FUNCTION_BLOCK RobotA21_1 EXTENDS KukaRobot
VAR_OUTPUT //from outputs array
	{warning disable C0195}
	//taskID : A21;
	//param1 : INT;
	//param2 : INT;
	//Xmm : INT;
	//Ymm : INT;
	//Zmm : INT;
	//angle : INT;
	//stagingOccupancy : INT;
	//insertionSuctionStatus : INT;
	//magazineStatus : INT; //unused
	inspectionValue : INT;
	
	strapSafetyOut : BOOL;
END_VAR
VAR_OUTPUT //from inputs array
	tool : SectionEnum := SectionEnum.WOOD_BUNK;
	suspendedMaterial : STRING;
	//gripper : EOAT := (id := SectionEnum.WOOD_BUNK, material := '');
	
	completedTask : A21;
	eoatDistance : INT;
	woodBunkAvailability : INT;
	chipboardAvailability : INT;
	materialAtHoldingPosition : INT;
	
	strapSafetyIn : BOOL;
END_VAR
VAR
	reservationEnum : SectionEnum;
	hmiTask : STRING;
	hmiTool : STRING;
END_VAR
(*
extends KukaRobot
assigns descriptive labels to each IO group from the array
additional section-specific methods to get/set IO groups
*)

(*
parameters - aliases to IO elements
command - full IO array
*)
{warning disable C0195}
SUPER^();

strapSafetyOut := NOT strapperA21.enable AND NOT strapperA21.execute;
outputs[8].15 := strapSafetyOut;

outputs[1] := taskID;
outputs[2] := param1;
outputs[3] := param2;
outputs[4] := Xmm;
outputs[5] := Ymm;
outputs[6] := Zmm;
outputs[7] := angle;
outputs[8] := stagingOccupancy;
outputs[9] := insertionSuctionStatus;
outputs[10] := magazineStatus;
outputs[11] := inspectionValue;

outputs[8].15 := strapSafetyOut;

refreshParameters();

reservationEnum := reservation;
IF reservationEnum = SectionEnum.NULL_SECTION THEN
	hmiReservation := 'N/A';
ELSE
	hmiReservation := TO_STRING(reservationEnum);
END_IF

hmiTask := TO_STRING(taskID);
hmiTool := TO_STRING(tool);

{attribute 'monitoring' := 'call'}
PROPERTY Angle : INT
GET
END_GET
SET
END_SET
END_PROPERTY

{attribute 'monitoring' := 'call'}
PROPERTY Busy : BOOL
GET
VAR
	//emptyOutput : ARRAY[1..50] OF INT;
END_VAR
//Busy stays TRUE until outputs are cleared AND completed task has elapsed
//Ready is always inverse of Busy
refreshParameters();

Busy := taskID <> 0 OR completedTask <> 0;
END_GET
END_PROPERTY

METHOD changeEOAT : BOOL
VAR_INPUT
	targetTool : SectionEnum;
END_VAR
setGroup(group := 1, value := A21.TOOL_CHANGE_CHIPBOARD);
setGroup(group := 1, value := A21.TOOL_CHANGE_BUNK);

changeEOAT := tool = targetTool;
END_METHOD

METHOD clearCommand : BOOL
VAR_INPUT
END_VAR
SUPER^.clearCommand();

refreshParameters();
END_METHOD

{attribute 'monitoring' := 'call'}
PROPERTY Done : BOOL
GET
refreshParameters();

Done :=
	completedTask = taskID AND
	taskID <> 0 AND
	completedTask <> 0;
END_GET
END_PROPERTY

{attribute 'monitoring' := 'call'}
PROPERTY HoldMaterial : STRING
GET
HoldMaterial := suspendedMaterial;
END_GET
SET
suspendedMaterial := HoldMaterial;
END_SET
END_PROPERTY

{attribute 'monitoring' := 'call'}
PROPERTY Param1 : INT
GET
END_GET
SET
END_SET
END_PROPERTY

{attribute 'monitoring' := 'call'}
PROPERTY Param2 : INT
GET
END_GET
SET
END_SET
END_PROPERTY

{attribute 'monitoring' := 'call'}
PROPERTY Ready : BOOL
GET
refreshParameters();

Ready := taskID = 0 AND completedTask = 0;
END_GET
END_PROPERTY

METHOD PRIVATE refreshParameters : BOOL
VAR_INPUT
END_VAR
{warning disable C0196}
taskID := outputs[1];
param1 := outputs[2];
param2 := outputs[3];
Xmm := outputs[4];
Ymm := outputs[5];
Zmm := outputs[6];
angle := outputs[7];
stagingOccupancy := outputs[8];
insertionSuctionStatus := outputs[9];
magazineStatus := outputs[10]; //unused
inspectionValue := outputs[11];

completedTask := inputs[1];
eoatDistance := inputs[2];
woodBunkAvailability := inputs[3];
chipboardAvailability := inputs[4];
materialAtHoldingPosition := inputs[5];
//robotEOAT := inputs[6];

strapSafetyIn := inputs[4].15;
END_METHOD

METHOD setGroup : BOOL
VAR_INPUT
	group : INT;
	value : INT;
END_VAR
SUPER^.setGroup(group := group, value := value);

refreshParameters();
END_METHOD

METHOD setParameters : BOOL
VAR_INPUT
	newTaskID : INT;
	newParam1 : INT;
	newParam2 : INT;
	newXmm : INT;
	newYmm : INT;
	newZmm : INT;
	newAngle : INT;
	newStagingOccupancy : INT;
	newInsertionSuctionStatus : INT;
	newMagazineStatus : INT; //unused
	newInspectionValue : INT;
END_VAR
setGroup(group := 1, value := newTaskID);
setGroup(group := 2, value := newParam1);
setGroup(group := 3, value := newParam2);
setGroup(group := 4, value := newXmm);
setGroup(group := 5, value := newYmm);
setGroup(group := 6, value := newZmm);
setGroup(group := 7, value := newAngle);

newStagingOccupancy.15 := NOT strapperA21.enable AND NOT strapperA21.execute;
setGroup(group := 8, value := newStagingOccupancy);

setGroup(group := 9, value := newInsertionSuctionStatus);
setGroup(group := 10, value := newMagazineStatus);
setGroup(group := 11, value := newInspectionValue);

refreshParameters();
END_METHOD

{attribute 'monitoring' := 'call'}
PROPERTY StagingOccupancy : INT
GET
END_GET
SET
END_SET
END_PROPERTY

{attribute 'monitoring' := 'call'}
PROPERTY TaskID : A21
GET
TaskID := outputs[1];
END_GET
SET
outputs[1] := TaskID;
END_SET
END_PROPERTY

{attribute 'monitoring' := 'call'}
PROPERTY Xmm : INT
GET
END_GET
SET
END_SET
END_PROPERTY

{attribute 'monitoring' := 'call'}
PROPERTY Ymm : INT
GET
END_GET
SET
END_SET
END_PROPERTY

{attribute 'monitoring' := 'call'}
PROPERTY Zmm : INT
GET
END_GET
SET
END_SET
END_PROPERTY

END_FUNCTION_BLOCK

(* stored: Version 1.1.0.1, ProductVersion 3.1.4024.11
   POU RobotA21_1: Id {67986ee9-35d0-4991-b5f7-67f7ce42987a}, SpecialFunc None
   Folder Groups: Id {eb42e132-aba5-47c8-8cae-a23ba92d8609}
   Folder Outputs: Id {321cea36-5d8f-400f-a5af-fdd868e827da}
   Folder Parameters: Id {c3d578fe-defd-4b12-9c77-b5953ca5c70d}
   Folder Properties: Id {eb91b964-775c-4fcb-b72d-754eac110c77}
   Property Angle: Id {4e283426-00f0-4c6b-b031-919967f9904b}
   Get Get: Id {86ab762a-e94a-42de-be5d-1c1d6883e23c}
   Set Set: Id {d8c9edf3-2c7c-45ce-acf1-984193f826aa}
   Property Busy: Id {79b3ce6a-9c01-452d-bb4a-867892b7100d}
   Get Get: Id {d9f24df2-3a79-4dc5-8239-3effa750f19a}
   Method changeEOAT: Id {056c48cb-6b24-46e5-adc1-74bf302c5ce2}
   Method clearCommand: Id {9155dabb-946e-465d-83be-8bd2e505d8d8}
   Property Done: Id {9e7360cb-1f33-47df-8e4b-f7735364d7f4}
   Get Get: Id {93f104fb-aef5-4ea5-b5b3-4fe7369ec6e3}
   Property HoldMaterial: Id {496f148f-ed6a-4218-9fd8-2d6729172b93}
   Get Get: Id {f10adf07-73d8-475e-92ad-0736f496bafa}
   Set Set: Id {6785f88a-284f-4b38-9b72-c0d119fc1118}
   Property Param1: Id {65d5818f-490f-4753-a4a0-b72affe7ebe5}
   Get Get: Id {33c584a1-59b3-4725-9a29-2b55d6bca155}
   Set Set: Id {a24ce27a-d8c3-4182-8d2d-af3bc85cb9c6}
   Property Param2: Id {45986bf8-e408-4761-908a-a14fdd4e0c5f}
   Get Get: Id {00d89721-8515-4692-bbde-4208e35fdac9}
   Set Set: Id {c3ea74de-9992-4db6-afa9-9cbc7c3fbab9}
   Property Ready: Id {369f7773-2368-4d49-8b91-351e545a75a3}
   Get Get: Id {215529ad-6487-4575-a731-48e5f5ac5cf5}
   Method refreshParameters: Id {84265115-d663-44b8-b8b9-61681c9d0c6b}
   Method setGroup: Id {611ab68f-21d7-4b39-adf2-beaae57f94ff}
   Method setParameters: Id {1354b4cc-1719-4f13-89cc-5f09b4fbd22b}
   Property StagingOccupancy: Id {9bae81f1-c5fb-4a8f-ad8e-8f4c91ef7270}
   Get Get: Id {723c3d8a-b1be-47c6-b0ec-da483ae38287}
   Set Set: Id {f470fa1e-412e-4fcf-85a7-315c141a0b58}
   Property TaskID: Id {102cf121-08b5-4ab1-acc2-91d63dc19216}
   Get Get: Id {e03ffefb-5ac7-4dff-833b-3d61f748f0a2}
   Set Set: Id {d2ad2f46-d6f2-4325-b62a-f39377561303}
   Property Xmm: Id {f8af782c-c8f6-493f-a864-cfc1423e1130}
   Get Get: Id {c16a2ea5-9b8c-4deb-9488-4660531b7328}
   Set Set: Id {cfb011be-897b-4911-a1d8-2244dac7b672}
   Property Ymm: Id {4c94e7f5-070a-4bf8-8d3a-ded0a4b2984e}
   Get Get: Id {30ca02e2-bb5f-4f31-a17e-3e1e0b4c77f6}
   Set Set: Id {bfd50408-c3b2-487a-99b7-c05c42200221}
   Property Zmm: Id {be5054f4-3eab-496c-b171-43999f2d1ea1}
   Get Get: Id {cb20c4c0-d3bd-41d3-9b78-0414a6ed1d9f}
   Set Set: Id {3b683ffd-7f40-4d22-a18b-70a17f375703} *)
